Fanuc KAREL source: kt00947.KL

-- PROVISIONAL review KL for V770-1; original PC SHA256 b8c2a3a6e985f793edff1d5af0fd9f77253162762f84e7a0d34221744b4d54ea
-- Incomplete behavior may be omitted. Consult companion uncertainty JSON. Do not deploy.
PROGRAM KT00947
%NOLOCKGROUP
VAR
  ENTRY : INTEGER
  PNAME : STRING[80]
  VNAME : STRING[80]
  STATUS : INTEGER
-- UNRESOLVED_DECL VALUE type=002012
BEGIN
  -- UNRESOLVED_PC offsets 5-12; opcodes 9C,23
  -- UNRESOLVED_PC offsets 17-25; opcodes 3F,75
  -- UNRESOLVED_PC offsets 30-43; opcodes 3F,75
  -- UNRESOLVED_PC offsets 48-86; opcodes 27,22,22,2A,22,2A,22,22,AF
  -- UNRESOLVED_PC offsets 91-95; opcodes 7F
END KT00947
